FUNCTION_BLOCK CHECKPOINT_DATA_SUBSCRIBER (* Composite Function Block Type *)
  (* Standard: 61499-2 *)
  (* Version 0.0, 12/17/2022, Dmitrii, Flexbridge AB, template *)
  PACKAGE UAO.Hackathon;
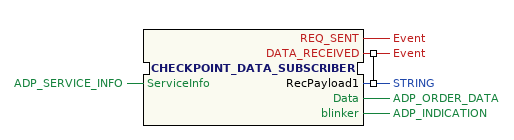
  EVENT_OUTPUT
    REQ_SENT;
    DATA_RECEIVED WITH RecPayload1;
  END_EVENT
  VAR_OUTPUT
    RecPayload1 : STRING;
  END_VAR
  SOCKETS
    ServiceInfo : ADP_SERVICE_INFO;
  END_SOCKETS
  PLUGS
    Data : ADP_ORDER_DATA;
    blinker : ADP_INDICATION;
  END_PLUGS
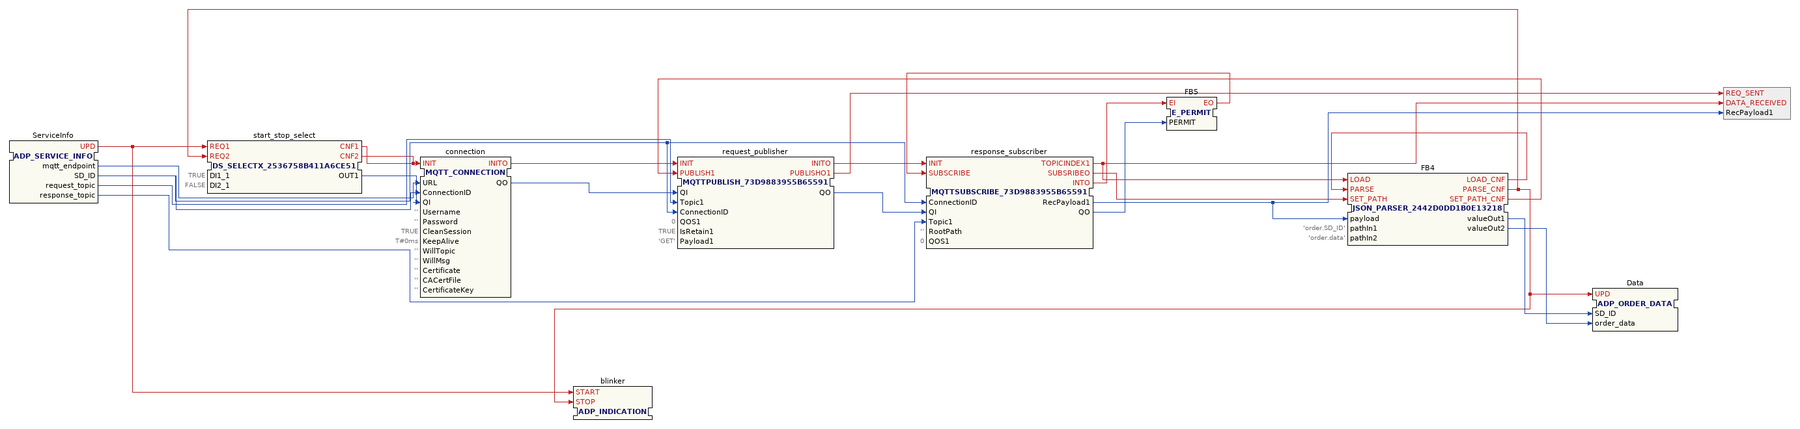
  FBS
    connection : MQTT_CONNECTION(Username := '', Password := '', CleanSession := TRUE, KeepAlive := T#0ms, WillTopic := '', WillMsg := '', Certificate := '', CACertFile := '', CertificateKey := '');
    response_subscriber : MQTTSUBSCRIBE_73D9883955B65591(RootPath := '', QOS1 := 0); {SET_ATTRIBUTE(Configuration.GenericFBType.InterfaceParams, nxtControl.CommProtocols#CNTX:=1)}
    FB4 : JSON_PARSER_2442D0DD1B0E13218(pathIn1 := 'order.SD_ID', pathIn2 := 'order.data'); {SET_ATTRIBUTE(Configuration.GenericFBType.InterfaceParams, Runtime.Base#CNT:=2;valueOut${CNT$}:STRING,STRING)}
    request_publisher : MQTTPUBLISH_73D9883955B65591(QOS1 := 0, IsRetain1 := TRUE, Payload1 := 'GET'); {SET_ATTRIBUTE(Configuration.GenericFBType.InterfaceParams, nxtControl.CommProtocols#CNTX:=1)}
    start_stop_select : DS_SELECTX_2536758B411A6CE51(DI1_1 := TRUE, DI2_1 := FALSE); {SET_ATTRIBUTE(Configuration.GenericFBType.InterfaceParams, Runtime.Standard#CNTX:=2;CNTY:=1;DI${CNTX,_,CNTY$}:BOOL)}
    FB5 : E_PERMIT;
  END_FBS
  EVENT_CONNECTIONS
    response_subscriber.TOPICINDEX1 TO FB4.LOAD;
    FB4.LOAD_CNF TO FB4.PARSE;
    FB4.PARSE_CNF TO Data.UPD;
    response_subscriber.SUBSRIBEO TO FB4.SET_PATH;
    connection.INITO TO request_publisher.INIT;
    request_publisher.INITO TO response_subscriber.INIT;
    response_subscriber.INTO TO FB5.EI;
    FB5.EO TO response_subscriber.SUBSCRIBE;
    ServiceInfo.UPD TO start_stop_select.REQ1;
    start_stop_select.CNF1 TO connection.INIT;
    start_stop_select.CNF2 TO connection.INIT;
    FB4.SET_PATH_CNF TO request_publisher.PUBLISH1;
    FB4.PARSE_CNF TO start_stop_select.REQ2;
    ServiceInfo.UPD TO blinker.START;
    FB4.PARSE_CNF TO blinker.STOP;
    request_publisher.PUBLISHO1 TO REQ_SENT;
    response_subscriber.TOPICINDEX1 TO DATA_RECEIVED;
  END_CONNECTIONS
  DATA_CONNECTIONS
    ServiceInfo.mqtt_endpoint TO connection.URL;
    ServiceInfo.SD_ID TO connection.ConnectionID;
    ServiceInfo.SD_ID TO response_subscriber.ConnectionID;
    response_subscriber.RecPayload1 TO FB4.payload;
    FB4.valueOut1 TO Data.SD_ID;
    FB4.valueOut2 TO Data.order_data;
    response_subscriber.QO TO FB5.PERMIT;
    start_stop_select.OUT1 TO connection.QI;
    connection.QO TO request_publisher.QI;
    request_publisher.QO TO response_subscriber.QI;
    ServiceInfo.request_topic TO request_publisher.Topic1;
    ServiceInfo.response_topic TO response_subscriber.Topic1;
    ServiceInfo.SD_ID TO request_publisher.ConnectionID;
    response_subscriber.RecPayload1 TO RecPayload1;
  END_CONNECTIONS
END_FUNCTION_BLOCK
